// TIA Portal V19 export
FUNCTION "IFM_PI1714_PD" : Void   // FC119, STL
TITLE = IFM PI1714 IO-Link Device Process Data
{ S7_Optimized_Access := 'TRUE' }
AUTHOR : AFL
FAMILY : IO_Link
NAME : PI1714PD
// This function reads device data for Pressure and Temperature
// and converts to physical units Bar and Â°C
//  ** If DeviceStatus = 4 then set Pressure_Bar to 20.0 and
//  Temperature_C to 200.0Â°C
// 
// Device status
// 0 (Everything is OK)
// 1 (Maintenance Required) 
// 2 (Out of specification)
// 3 (Functional check)
// 4 (Failure)
//  ********************************************************
// stored: AutoNumber false
   VAR_INPUT
      Addr : Int;   // First Byte address of 12 + PQI byte address space
   END_VAR
   VAR_OUTPUT
      Pressure_Bar : Real;   // Current Valve (-10000 to 168000) * 0.0001
      Temperature_C : Real;   // Current Valve (-3000 to 16000) * 0.01
      DeviceStatus : Byte;   // See Block Comment
      OUT2 : Bool;   // Current status of DO OUT2
      OUT1 : Bool;   // Current status of DO OUT1
      O_DI4 : Bool;   // Output signal status Pin 4
      O_DI2 : Bool;   // Output signal status Pin 2
      O_DA : Bool;   // Output device recognised
      O_DE : Bool;   // Output device error event has appeared
      O_PQ : Bool;   // Output port qualifer proces data valid VAR_IN_OUT END_VAR
   END_VAR
   VAR_TEMP
      TW_Flag : Word;
      Tmp_word : Word;   // LW2
   END_VAR
BEGIN

NETWORK
TITLE = 
// Get first byte address
      L     #Addr;
      SLW   3;
      LAR1;
// **************  Inputs *******************
// Pressure converted to Bar
      L     ID [AR1, P#0.0];
      DTR;
      L     0.0001;
      *R;
      T     #Pressure_Bar;
// Temperature converted to Bar
      L     ID [AR1, P#6.0];
      DTR;
      L     0.01;
      *R;
      T     #Temperature_C;

// Device Status
      L     IW [AR1, P#10.0];
      T     #Tmp_word;
      L     16#00F0;  //Clear OUT2 and OUT1 bits and temp scale byte
      AW;
      T     #Tmp_word;
      SRW   4;
      T     #Tmp_word;
      L     #Tmp_word.%B0;
      T     #DeviceStatus;
//See block comment for value meanings


// PQI

      L     IB [AR1, P#12.0];
      T     #TW_Flag;

      L     #TW_Flag;
      L     1;
      AW;
      L     1;
      ==I;
      =     #O_DI4;



      L     #TW_Flag;
      L     2;
      AW;
      L     2;
      ==I;
      =     #O_DI2;

      L     #TW_Flag;
      L     32;
      AW;
      L     32;
      ==I;
      =     #O_DA;

      L     #TW_Flag;
      L     64;
      AW;
      L     64;
      ==I;
      =     #O_DE;


      L     #TW_Flag;
      L     128;
      AW;
      L     128;
      ==I;
      =     #O_PQ;

// *** Fail High ***
      L     #DeviceStatus;
      L     4;
      ==I;
      JCN   END;
      L     20.0;
      T     #Pressure_Bar;
      L     200.0;
      T     #Temperature_C;
END:  NOP   0;
END_FUNCTION
